//{attribute 'qualified_only'}
{attribute 'strict'}
TYPE eOrMethod :
(
	Maximum
);
END_TYPE

(* stored: Version 1.1.0.1, ProductVersion 3.1.4024.6
   DUT eOrMethod: Id {cc8a16c5-66a3-4ea1-9aba-14c8504f75db} *)
